INTERFACE I_Axis

END_INTERFACE

(* stored: Version 1.1.0.1, ProductVersion 3.1.4024.12
   Itf I_Axis: Id {d6375579-dabd-45c1-b30f-cdc924ac59c7} *)
